TYPE AxesUnlockBrakeProcessArgs :
STRUCT
	///Unlock the brake for this number of seconds (0 means forever)
	seconds: LREAL := 10.0;
END_STRUCT
END_TYPE

(* stored: Version 1.1.0.1, ProductVersion 3.1.4019.2
   DUT AxesUnlockBrakeProcessArgs: Id {51322f4d-d17e-4c91-a375-2ec7f1785cf4} *)
